FUNCTION AsTag : Result
VAR_INPUT
	iSource	: I_Component;
END_VAR
VAR_OUTPUT
	iDest	: I_Tag;
END_VAR

IF iSource = 0 THEN
	AsTag := Err.Itf0;
	RETURN;
END_IF

IF __QUERYINTERFACE(iSource, iDest) THEN
	AsTag := Ok;
ELSE
	AsTag := Err.NoMatch;
END_IF

END_FUNCTION

(* stored: Version 1.1.0.1
   POU AsTag: Id {3feb1b07-c695-429c-b10c-285305651b80}, SpecialFunc None *)
